FUNCTION tempSAFE : BOOL
VAR_INPUT
	TEMPcel : INT;
	thresholdTEMPcel : INT;
END_VAR
VAR
END_VAR

// If temp passed is under threshold, returns TRUE (is safe)
IF TEMPcel <= thresholdTEMPcel THEN
	tempSAFE := TRUE;
ELSE 
	tempSAFE := FALSE;
END_IF;

END_FUNCTION

(* stored: Version 1.1.0.1, ProductVersion 3.1.4024.9
   POU tempSAFE: Id {1b5d8ed3-56fd-47e7-8f93-54d863623bfe}, SpecialFunc None *)
